(* IEC 61131-3 sources: NVM-AquaFeed-Platform/02_Software_Design/PLC/07_Implementation/Functions, 2 files *)

(* ---- F_CyclicDistance.st ---- *)
FUNCTION F_CyclicDistance : DINT
VAR_INPUT
    diCurrentPosition : DINT;
    diTargetPosition : DINT;
    diCycleLength : DINT;
END_VAR
VAR
    diForwardDistance : DINT;
    diReverseDistance : DINT;
END_VAR

diForwardDistance := diTargetPosition - diCurrentPosition;
IF diForwardDistance < 0 THEN
    diForwardDistance := diForwardDistance + diCycleLength;
END_IF;

diReverseDistance := diCurrentPosition - diTargetPosition;
IF diReverseDistance < 0 THEN
    diReverseDistance := diReverseDistance + diCycleLength;
END_IF;

IF diForwardDistance <= diReverseDistance THEN
    F_CyclicDistance := diForwardDistance;
ELSE
    F_CyclicDistance := diReverseDistance;
END_IF;

END_FUNCTION

(* ---- F_ElapsedMs.st ---- *)
FUNCTION F_ElapsedMs : UDINT
VAR_INPUT
    udiCurrentTickMs : UDINT;
    udiStartTickMs : UDINT;
END_VAR

IF udiCurrentTickMs >= udiStartTickMs THEN
    F_ElapsedMs := udiCurrentTickMs - udiStartTickMs;
ELSE
    F_ElapsedMs := (c_udiCounterMaximum - udiStartTickMs) +
                   udiCurrentTickMs + 1;
END_IF;

END_FUNCTION
